PROGRAM PRG_Compilation
VAR
	senNO				: FB_Sensor_NO;
	senNO_DecoratorTest	: FB_Sensor_NO_TestDecorator (fbToDecorate := senNO);
	senNC				: FB_Sensor_NC;
	senNC_DecoratorTest	: FB_Sensor_NC_TestDecorator (fbToDecorate := senNC);
	sen2NO				: FB_Sensor_NO_2InRow;
	sen2NO_DecoratorTest: FB_Sensor_NO_2InRow_TestDecorator (fbToDecorate := sen2NO);
	
END_VAR

END_PROGRAM

(* stored: Version 1.1.0.1
   POU PRG_Compilation: Id {fee939fc-f789-4718-9ef1-7cf0d54cde09}, SpecialFunc None *)
